FUNCTION_BLOCK "EM_Outled"
{ S7_Optimized_Access := 'TRUE' }


BEGIN

END_FUNCTION_BLOCK
